// TwinCAT 3 PLC project FMMath
// Title: FM Math
// Company: FrameworkMonorepo
// ProjectVersion: 0.0.1
// ProgramVersion: 3.1.4024.0
// libraries:
//   Tc2_Math, * (Beckhoff Automation GmbH)
// project tree:
//   Fraction/ Fraction.TcDUT
//   Arithmetic/ ModuloLREAL.TcPOU, Pow2.TcPOU, Pow3.TcPOU
//   Point/Equals/ EqualsLREAL.TcPOU, EqualsPoint2D.TcPOU, EqualsPoint3D.TcPOU
//   Point/ Point3D.TcDUT, Point2D.TcDUT
//   Range/Equals/ EqualsRange.TcPOU
//   Range/IsInRange/ IsInRangeInclusive.TcPOU, IsInRangeInclusive2D.TcPOU, IsInRangeInclusive3D.TcPOU
//   Range/ Range2D.TcDUT, Range3D.TcDUT, Range.TcDUT
//   Version/ Global_Version.TcGVL
// (motion and I/O tree: see PLC project fmtypes)
// real-time tasks:
//   TASK BindingTestTask: cycle T#1ms, priority 20, ADS port 350
//   TASK PlcTask: cycle T#1ms, priority 21, ADS port 351
//   TASK PlcTask1: cycle T#1ms, priority 22, ADS port 352
//   TASK PlcTask2: cycle T#1ms, priority 23, ADS port 353
//   TASK MathTestTask: cycle T#1ms, priority 24, ADS port 354
//   TASK TimesTestsTask: cycle T#1ms, priority 25, ADS port 355

// ---- Fraction/Fraction.TcDUT
TYPE Fraction :
STRUCT
	Numerator : LREAL;
	Denominator : LREAL;
END_STRUCT
END_TYPE

// ---- Point/Point3D.TcDUT
TYPE Point3D :
STRUCT
	X : LREAL;
	Y : LREAL;
	Z : LREAL;
END_STRUCT
END_TYPE

// ---- Point/Point2D.TcDUT
TYPE Point2D :
STRUCT
	X : LREAL;
	Y : LREAL;
END_STRUCT
END_TYPE

// ---- Range/Range2D.TcDUT
TYPE Range2D :
STRUCT
	X : Range;
	Y : Range;
END_STRUCT
END_TYPE

// ---- Range/Range3D.TcDUT
TYPE Range3D :
STRUCT
	X : Range;
	Y : Range;
	Z : Range;
END_STRUCT
END_TYPE

// ---- Range/Range.TcDUT
TYPE Range :
STRUCT
	Bottom : LREAL;
	Top : LREAL;
END_STRUCT
END_TYPE

// ---- Version/Global_Version.TcGVL
{attribute 'TcGenerated'}
{attribute 'no-analysis'}
{attribute 'linkalways'}
// This function has been automatically generated from the project information.
VAR_GLOBAL CONSTANT
	{attribute 'const_non_replaced'}
	stLibVersion_FM_Math : ST_LibVersion := (iMajor := 0, iMinor := 0, iBuild := 1, iRevision := 0, nFlags := 0, sVersion := '0.0.1');
END_VAR

// ---- Arithmetic/ModuloLREAL.TcPOU
FUNCTION ModuloLREAL : LREAL
VAR_INPUT
	divident : LREAL;
	modulus : LREAL;
END_VAR

ModuloLREAL := divident - modulus * FLOOR(divident / modulus);

END_FUNCTION

// ---- Arithmetic/Pow2.TcPOU
FUNCTION Pow2 : LREAL
VAR_INPUT
	number : LREAL;
END_VAR

Pow2 := number * number;

END_FUNCTION

// ---- Arithmetic/Pow3.TcPOU
FUNCTION Pow3 : LREAL
VAR_INPUT
	number : LREAL;
END_VAR

Pow3 := number * number * number;

END_FUNCTION

// ---- Point/Equals/EqualsLREAL.TcPOU
FUNCTION EqualsLREAL : BOOL
VAR_INPUT
	n1 : LREAL;
	n2 : LREAL;
	epsilon : LREAL;
END_VAR

EqualsLREAL := ABS(n1 - n2) <= epsilon;

END_FUNCTION

// ---- Point/Equals/EqualsPoint2D.TcPOU
FUNCTION EqualsPoint2D : BOOL
VAR_INPUT
	p1 : Point2D;
	p2 : Point2D;
	epsilon : Point2D;
END_VAR

EqualsPoint2D := EqualsLREAL(p1.X, p2.X, epsilon.X)
			AND EqualsLREAL(p1.Y, p2.Y, epsilon.Y);

END_FUNCTION

// ---- Point/Equals/EqualsPoint3D.TcPOU
FUNCTION EqualsPoint3D : BOOL
VAR_INPUT
	p1 : Point3D;
	p2 : Point3D;
	epsilon : Point3D;
END_VAR

EqualsPoint3D := EqualsLREAL(p1.X, p2.X, epsilon.X)
			AND EqualsLREAL(p1.Y, p2.Y, epsilon.Y)
			AND EqualsLREAL(p1.Z, p2.Z, epsilon.Z);

END_FUNCTION

// ---- Range/Equals/EqualsRange.TcPOU
FUNCTION EqualsRange : BOOL
VAR_INPUT
	range1 : Range;
	range2 : Range;
	epsilon : LREAL;
END_VAR

EqualsRange := EqualsLREAL(range1.Bottom, range2.Bottom, epsilon)
			AND EqualsLREAL(range1.Top, range2.Top, epsilon);

END_FUNCTION

// ---- Range/IsInRange/IsInRangeInclusive.TcPOU
FUNCTION IsInRangeInclusive : BOOL
VAR_INPUT
	value : LREAL;
	range : Range;
END_VAR

IsInRangeInclusive := range.Bottom <= value AND value <= range.Top;

END_FUNCTION

// ---- Range/IsInRange/IsInRangeInclusive2D.TcPOU
FUNCTION IsInRangeInclusive2D : BOOL
VAR_INPUT
	point : Point2D;
	range : Range2D;
END_VAR

IsInRangeInclusive2D := 
	IsInRangeInclusive(point.X, range.X)
	AND IsInRangeInclusive(point.Y, range.Y)
	;

END_FUNCTION

// ---- Range/IsInRange/IsInRangeInclusive3D.TcPOU
FUNCTION IsInRangeInclusive3D : BOOL
VAR_INPUT
	point : Point3D;
	range : Range3D;
END_VAR

IsInRangeInclusive3D := 
	IsInRangeInclusive(point.X, range.X)
	AND IsInRangeInclusive(point.Y, range.Y)
	AND IsInRangeInclusive(point.Z, range.Z)
	;

END_FUNCTION
